KUKA KRL program: TTT_Kreis.src, TTT_Kreis.dat

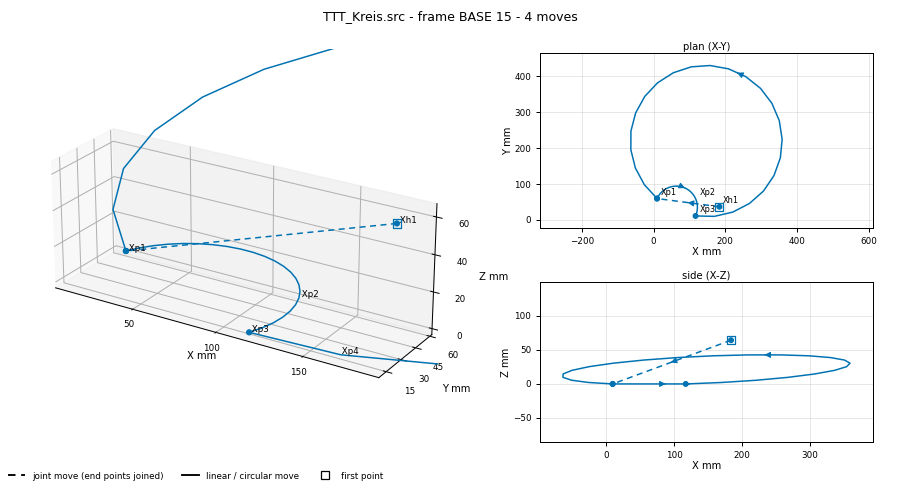
[picture p0: tool path of TTT_Kreis.src in frame BASE 15, 4 of 6 moves have a stored position in this frame; points joined in program order, loops and branches not executed]
--- TTT_Kreis.src ---
&ACCESS RVO1
&COMMENT
DEF TTT_Kreis ( )
;FOLD INI
  ;FOLD BASISTECH INI
    GLOBAL INTERRUPT DECL 3 WHEN $STOPMESS==TRUE DO IR_STOPM ( )
    INTERRUPT ON 3
    BAS (#INITMOV,0 )
  ;ENDFOLD (BASISTECH INI)
  ;FOLD USER INI
    ;Make your modifications here

  ;ENDFOLD (USER INI)
;ENDFOLD (INI)

;FOLD PTP HOME  Vel= 100 % DEFAULT;%{PE}%MKUKATPBASIS,%CMOVE,%VPTP,%P 1:PTP, 2:HOME, 3:, 5:100, 7:DEFAULT
$BWDSTART = FALSE
PDAT_ACT=PDEFAULT
FDAT_ACT=FHOME
BAS (#PTP_PARAMS,100 )
$H_POS=XHOME
PTP  XHOME
;ENDFOLD

;FOLD PTP h1 CONT Vel=100 % PDAT8 Tool[15] Base[15];%{PE}%R 8.3.22,%MKUKATPBASIS,%CMOVE,%VPTP,%P 1:PTP, 2:h1, 3:C_PTP, 5:100, 7:PDAT8
$BWDSTART=FALSE
PDAT_ACT=PPDAT8
FDAT_ACT=Fh1
BAS(#PTP_PARAMS,100)
PTP Xh1 C_PTP
;ENDFOLD

;FOLD PTP p1  Vel=100 % PDAT9 Tool[15] Base[15];%{PE}%R 8.3.22,%MKUKATPBASIS,%CMOVE,%VPTP,%P 1:PTP, 2:p1, 3:, 5:100, 7:PDAT9
$BWDSTART=FALSE
PDAT_ACT=PPDAT9
FDAT_ACT=Fp1
BAS(#PTP_PARAMS,100)
PTP Xp1
;ENDFOLD

;FOLD CIRC p2 p3  Vel=1 m/s CPDAT13 Tool[15] Base[15];%{PE}%R 8.3.22,%MKUKATPBASIS,%CMOVE,%VCIRC,%P 1:CIRC, 2:p2, 3:p3, 4:, 6:1, 8:CPDAT13
$BWDSTART=FALSE
LDAT_ACT=LCPDAT13
FDAT_ACT=Fp3
BAS(#CP_PARAMS,1)
CIRC Xp2, Xp3
;ENDFOLD

;FOLD CIRC p4 p1  Vel=1 m/s CPDAT14 Tool[15] Base[15];%{PE}%R 8.3.22,%MKUKATPBASIS,%CMOVE,%VCIRC,%P 1:CIRC, 2:p4, 3:p1, 4:, 6:1, 8:CPDAT14
$BWDSTART=FALSE
LDAT_ACT=LCPDAT14
FDAT_ACT=Fp1
BAS(#CP_PARAMS,1)
CIRC Xp4, Xp1
;ENDFOLD

;FOLD PTP HOME  Vel= 100 % DEFAULT;%{PE}%MKUKATPBASIS,%CMOVE,%VPTP,%P 1:PTP, 2:HOME, 3:, 5:100, 7:DEFAULT
$BWDSTART = FALSE
PDAT_ACT=PDEFAULT
FDAT_ACT=FHOME
BAS (#PTP_PARAMS,100 )
$H_POS=XHOME
PTP  XHOME
;ENDFOLD

END

--- TTT_Kreis.dat ---
&ACCESS RVO1
&COMMENT
DEFDAT TTT_Kreis PUBLIC
;FOLD EXTERNAL DECLARATIONS;%{PE}%MKUKATPBASIS,%CEXT,%VCOMMON,%P
;FOLD BASISTECH EXT;%{PE}%MKUKATPBASIS,%CEXT,%VEXT,%P
EXT  BAS (BAS_COMMAND  :IN,REAL  :IN )
DECL INT SUCCESS
;ENDFOLD (BASISTECH EXT)
;FOLD USER EXT;%{E}%MKUKATPUSER,%CEXT,%VEXT,%P
;Make here your modifications

;ENDFOLD (USER EXT)
;ENDFOLD (EXTERNAL DECLERATIONS)
DECL INT scale=1
DECL BASIS_SUGG_T LAST_BASIS={POINT1[] "p4",POINT2[] "p1",CP_PARAMS[] "CPDAT14",PTP_PARAMS[] "PDAT9",CONT[] "",CP_VEL[] "1",PTP_VEL[] "100"}
DECL E6POS Xh1={X 183.741989,Y 36.8539124,Z 64.0154648,A -16.3441830,B 34.6527901,C -162.031189,S 2,T 3,E1 0.0,E2 0.0,E3 0.0,E4 0.0,E5 0.0,E6 0.0}
DECL FDAT Fh1={TOOL_NO 15,BASE_NO 15,IPO_FRAME #BASE,POINT2[] " ",TQ_STATE FALSE}
DECL PDAT PPDAT8={VEL 100,ACC 100,APO_DIST 100,APO_MODE #CPTP,GEAR_JERK 50}
DECL E6POS Xp1={X 9.81686211,Y 59.8364639,Z -0.258725,A -121.950264,B 87.5867615,C 47.4774323,S 2,T 2,E1 0.0,E2 0.0,E3 0.0,E4 0.0,E5 0.0,E6 0.0}
DECL FDAT Fp1={TOOL_NO 15,BASE_NO 15,IPO_FRAME #BASE,POINT2[] "p1",TQ_STATE FALSE}
DECL PDAT PPDAT9={VEL 100,ACC 100,APO_DIST 100,APO_MODE #CPTP,GEAR_JERK 50}
DECL E6POS Xp2={X 117.147263,Y 59.8364639,Z -0.258725524,A -121.950256,B 87.5867615,C 47.4774323,S 2,T 35,E1 0.0,E2 0.0,E3 0.0,E4 0.0,E5 0.0,E6 0.0}
DECL E6POS Xp3={X 117.158791,Y 11.2463903,Z -0.276550800,A -121.976845,B 87.5970078,C 47.4512978,S 2,T 3,E1 0.0,E2 0.0,E3 0.0,E4 0.0,E5 0.0,E6 0.0}
DECL FDAT Fp3={TOOL_NO 15,BASE_NO 15,IPO_FRAME #BASE,POINT2[] "p3",TQ_STATE FALSE}
DECL LDAT LCPDAT13={VEL 1,ACC 100,APO_DIST 100,APO_FAC 50,AXIS_VEL 100.0,AXIS_ACC 100.0,ORI_TYP #VAR,CIRC_TYP #BASE,JERK_FAC 50.0,GEAR_JERK 50.0,EXAX_IGN 0}
DECL E6POS Xp4={X 168.454956,Y 10.0288706,Z 1.79486394,A -16.3441811,B 34.6527901,C -162.031189,S 2,T 3,E1 0.0,E2 0.0,E3 0.0,E4 0.0,E5 0.0,E6 0.0}
DECL LDAT LCPDAT14={VEL 1,ACC 100,APO_DIST 100,APO_FAC 50,AXIS_VEL 100.0,AXIS_ACC 100.0,ORI_TYP #VAR,CIRC_TYP #BASE,JERK_FAC 50.0,GEAR_JERK 50.0,EXAX_IGN 0}
ENDDAT
